// TIA Portal V18 export
DATA_BLOCK "IEC_Counter_0_DB"   // DB139
{ S7_Optimized_Access := 'TRUE' }
// stored: AutoNumber true, DBAccessibleFromOPCUA true, InstanceOfName IEC_UDCOUNTER, OfSystemLibElement IEC_UDCOUNTER, OfSystemLibVersion 1.0
"IEC_UDCOUNTER"
   // VAR RETAIN
   //    CU : Bool;
   //    CD : Bool;
   //    R : Bool;
   //    LD : Bool;
   //    QU : Bool;
   //    QD : Bool;
   //    PV : UDInt;
   //    CV : UDInt;
   // END_VAR
BEGIN
END_DATA_BLOCK
